FUNCTION_BLOCK fbSimSCA
VAR_INPUT
	CommandSpeedRaw : DINT;
	CommandDir : BOOL; // 1 = Forward, 0 = Backward
END_VAR
VAR_OUTPUT
	ActualSpeedRaw : DINT;
	ActualDir : BOOL; // 1 = Forward, 0 = Backward
END_VAR
VAR
	Acceleration : DINT := 10; // defines the spead change per PLC cycle time
	CommandSpeed: DINT;
	ActualSpeed: DINT := 0;
END_VAR

IF CommandDir THEN
	CommandSpeed := CommandSpeedRaw;
ELSE
	CommandSpeed := -CommandSpeedRaw;
END_IF

IF ActualSpeed > 0 THEN
	ActualDir := 1;
	ActualSpeedRaw := ActualSpeed;
ELSE
	ActualDir := 0;
	ActualSpeedRaw := -ActualSpeed;
END_IF

IF ActualSpeed < CommandSpeed - Acceleration THEN
	ActualSpeed := ActualSpeed + Acceleration;
END_IF

IF ActualSpeed > CommandSpeed + Acceleration THEN
	ActualSpeed := ActualSpeed - Acceleration;
END_IF

IF ActualSpeed >= CommandSpeed - Acceleration AND ActualSpeed <= CommandSpeed + Acceleration THEN
	ActualSpeed := CommandSpeed;
END_IF

END_FUNCTION_BLOCK

(* stored: Version 1.1.0.1, ProductVersion 3.1.4022.17
   POU fbSimSCA: Id {635c4bfd-7d02-4ee1-90b4-bcd6764906c4}, SpecialFunc None *)
